(* IEC 61131-3 sources: moqui-plc/iec61131/moqui/runtime/component/mantle-hvac/src/main/org/moqui/device, 14 files *)

(* ---- AirDistributionControllerStatus.st ---- *)
TYPE AirDistributionControllerStatus : (
    Init := 0,
    HighPhase,
    TransitionToLow,
    LowPhase,
    TransitionToHigh
); END_TYPE

(* ---- DeviceFacade.dut ---- *)
(*#-#-#-#-#-#-#-#-#-#---Declaration---#-#-#-#-#-#-#-#-#-#-#-#-#*)

(*
 * DeviceFacade implementation for managing devices and logical parameters.
 *
 * Naming rules:
 *   deviceName + parameterName or parameterName → logical signal
 *   deviceName + parameterName or parameterName + Min/Max → limits
 *
 * All digital signals (boolean) are active-high (positive logic).
 * All durations are expressed in seconds TUnit.
 *)
TYPE DeviceFacade : STRUCT
	(* HVAC process control parameters (setpoints, limits, etc.) and process sensor signals *)
    (* Cell T+RH sensor  *)
    (* Setpoints and limits - mapped from recipe *)
    tempSetpoint : REAL; (* °C target process temperature *)
    tempHysteresis : REAL; (* °C symmetric hysteresis band *)
    tempMin : REAL;   (* °C absolute lower limit (alarm) *)
    tempMax : REAL; (* °C absolute upper limit (alarm) *)
    rhSetpoint : REAL; (* %  target relative humidity *)
    rhHysteresis : REAL; (* %  symmetric hysteresis band *)
    rhMin : REAL; (* % lower limit *)
    rhMax : REAL; (* % upper limit *)
    (* Core / surface probes - optional, used for thawing phases *)
    tempCoreSetpoint : REAL;
    tempCoreHysteresis : REAL;
    tempSurfaceSetpoint : REAL;
    tempSurfaceHysteresis : REAL;
    tempSurfaceMax : REAL;

    (* Feedback - wired from InputSignalUpdate each scan *)
    tempFeedback : REAL; (* °C cell air temperature *)
    rhFeedback : REAL; (* % cell relative humidity *)
    tempCoreFeedback : REAL; (* °C product core temperature *)
    tempSurfaceFeedback : REAL; (* °C product surface temperature *)

    (* Duct T+RH sensor (probe in the pipes) *)
    (* Limits - mapped from recipe or fixed commissioning values *)
    ductTempMin : REAL; (* °C minimum safe supply-air temperature *)
    ductTempMax : REAL; (* °C maximum safe supply-air temperature *)
    ductRhMax : REAL; (* % maximum allowed supply-air humidity *)
    (* Feedback - wired from InputSignalUpdate each scan *)
    ductTempFeedback : REAL; (* °C supply-air temperature in duct *)
    ductRhFeedback : REAL; (* % supply-air relative humidity in duct *)

    (* Boolean predicates - computed each scan by MainRuleEngine *)
    (* Cell sensor *)
    tempInRange : BOOL; (* tempMin+hys ≤ T ≤ tempMax-hys *)
    tempAtSetpoint : BOOL; (* |T - Tsp| ≤ hys *)
    tempOverMax : BOOL; (* T > tempMax *)
    tempOverMin : BOOL; (* T > tempMin *)
    tempUnderMin : BOOL; (* T < tempMin *)
    tempUnderMax : BOOL; (* T < tempMax *)
    tempCoreAtSetpoint : BOOL;
    tempSurfaceAtSetpoint : BOOL;
    tempSurfaceOverMax : BOOL;
    tempSurfaceUnderMax : BOOL;
    rhAtSetpoint : BOOL;
    rhOverMax  : BOOL; (* RH > rhMax - hys *)
    rhUnderMin : BOOL; (* RH < rhMin + hys *)
    rhOverMin : BOOL;
    rhUnderMax : BOOL;
    (* Duct sensor - safety predicates *)
    ductTempOverMax : BOOL; (* Supply air too hot → product at risk  *)
    ductTempUnderMin : BOOL; (* Supply air too cold → product at risk  *)
    ductRhOverMax : BOOL; (* Supply air saturated → condensation risk *)

    (* Operating-mode flags and process timing (mapped from recipe). *)
    rhControlEnabled : BOOL; (* Cooling+Heating both active for RH ctrl *)
    rhControlOnly : BOOL; (* Stop when RH ≤ rhMin regardless of time *)
    tempCoreControlEnabled : BOOL; (* Use core probe for thawing end-of-phase *)
    airMixingEnabled : BOOL;
    (* Process cycle durations (seconds) *)
    processEstimatedDuration : UDINT;
    processMinDuration : UDINT;
    processActualDuration : UDINT;
    processRemainingDuration : UDINT;
    (* Process time tracking *)
    (* Run / break cycle - phase 4 *)
    estimatedRuntime : UDINT;
    minRuntime : UDINT;
    actualRuntime : UDINT;
    estimatedBreakDuration : UDINT;
    minBreakDuration : UDINT;
    actualBreakDuration : UDINT;
    (* Air mixing sub-cycle *)
    airMixingEstimatedDuration : UDINT;
    airMixingMinDuration : UDINT;
    airMixingActualDuration : UDINT;
    airMixingEstimatedBreakDuration : UDINT;
    airMixingMinBreakDuration : UDINT;
    airMixingActualBreakDuration : UDINT;
    (* Flags *)
    (*
     * For operations based on equalization phases, rest/recovery periods are used,
     * during which moisture is evenly redistributed between the core
     * and the surface of the product after an intense drying phase (pulling).
     *)
    timeBreakEnabled : BOOL; (* TRUE while in break period *)
    isCompleted : BOOL; (* TRUE when the work effort is finished *)

    (* Main FSM state and transition request/acknowledge commands *)
    status : MainStatus := MainStatus.Standby;
    lastStatus : MainStatus := MainStatus.Standby;
    (*
     * Internally generated transition requests (set by MainRuleEngine,
     * consumed and cleared by Main.pou each scan)
     *)
    standbyRequest : BOOL;
    ventilationRequest : BOOL;
    coolingRequest : BOOL;
    heatingRequest : BOOL;
    dryingRequest : BOOL;
    surfaceThawingRequest : BOOL;
    coreThawingRequest : BOOL;
    faultRequest : BOOL;
    resetRequest : BOOL;

    (* HVAC devices *)

    (* Cold glycol group *)
    (* Enable/disable requests: written by Main component, read by DeviceManager *)
    coldGroupEnableRequest : BOOL;
    coldGroupDisableRequest : BOOL;
    (* Glycol circulating pump - on/off Actuator *)
    coldGlycolPump : Actuator;
    (* Modulating glycol valve - continuous PID control *)
    coldGlycolValve : ProcessPid;

    (* Hot glycol group *)
    hotGroupEnableRequest : BOOL;
    hotGroupDisableRequest : BOOL;
    hotGlycolPump : Actuator;
    hotGlycolValve : ProcessPid;

    (* AHU fan *)
    ahuFanEnableRequest : BOOL;
    (* Speed setpoint (0.0 … 100.0 %) - from recipe *)
    ahuFanSpeedSetpoint : REAL;
    (* Speed feedback (0.0 … 100.0 %) - from InputSignalUpdate *)
    ahuFanSpeedFeedback : REAL;
    ahuFan : ProcessPid;

    (* Air-flow distributor *)
    (* Treated as Actuator with additional ref/feedback.
     * The drive alternates air distribution between left and right ducts.
     * ref = time-split setpoint (0-100 %, 0 = full left, 100 = full right).
     * feedback = actual drive speed feedback.
	 *)
    airFlowEnableRequest : BOOL;
    airFlowDisableRequest : BOOL;
    airFlowRef : REAL; (* duty-cycle / distribution setpoint *)
    airFlowSpeedFeedback : REAL; (* drive speed feedback *)
    airFlow : Actuator;

    (* Signal management - centralised fault / alarm / warning engine *)
    signalMgmt : SignalMgmt;
END_STRUCT END_TYPE

(* ---- DeviceFacade.st ---- *)
(*
 * DeviceFacade implementation for managing devices and logical parameters.
 *
 * Naming rules:
 *   deviceName + parameterName or parameterName -> logical signal
 *   deviceName + parameterName or parameterName + Min/Max -> limits
 *
 * All digital signals (boolean) are active-high (positive logic).
 * All durations are expressed in seconds TUnit.
 *)
TYPE DeviceFacade : STRUCT
	(* HVAC process control parameters (setpoints, limits, etc.) and process sensor signals *)
    (* Cell T+RH sensor  *)
    (* Setpoints and limits - mapped from recipe *)
    tempSetpoint : REAL; (* °C target process temperature *)
    tempHysteresis : REAL; (* °C symmetric hysteresis band *)
    tempMin : REAL;   (* °C absolute lower limit (alarm) *)
    tempMax : REAL; (* °C absolute upper limit (alarm) *)
    rhSetpoint : REAL; (* %  target relative humidity *)
    rhHysteresis : REAL; (* %  symmetric hysteresis band *)
    rhMin : REAL; (* % lower limit *)
    rhMax : REAL; (* % upper limit *)
    (* Feedback - wired from InputSignalUpdate each scan *)
    tempFeedback : REAL; (* °C zone air temperature *)
    rhFeedback : REAL; (* % zone relative humidity *)

    (* Duct T+RH sensor (probe in the pipes) *)
    (* Limits - mapped from recipe or fixed commissioning values *)
    ductTempMin : REAL; (* °C minimum safe supply-air temperature *)
    ductTempMax : REAL; (* °C maximum safe supply-air temperature *)
    ductRhMax : REAL; (* % maximum allowed supply-air humidity *)
    (* Feedback - wired from InputSignalUpdate each scan *)
    ductTempFeedback : REAL; (* °C supply-air temperature in duct *)
    ductRhFeedback : REAL; (* % supply-air relative humidity in duct *)

    (* Boolean predicates - computed each scan by MainRuleEngine *)
    (* Cell sensor *)
    tempInRange : BOOL; (* tempMin+hys <= T <= tempMax-hys *)
    tempAtSetpoint : BOOL; (* |T - Tsp| <= hys *)
    tempAboveSetpointBand : BOOL; (* T >= tempSetpoint + tempHysteresis *)
    tempBelowSetpointBand : BOOL; (* T <= tempSetpoint - tempHysteresis *)
    tempOverMax : BOOL; (* T > tempMax *)
    tempOverMin : BOOL; (* T > tempMin *)
    tempUnderMin : BOOL; (* T < tempMin *)
    tempUnderMax : BOOL; (* T < tempMax *)
    rhAtSetpoint : BOOL;
    rhOverMax  : BOOL; (* RH > rhMax - hys *)
    rhUnderMin : BOOL; (* RH < rhMin + hys *)
    rhOverMin : BOOL;
    rhUnderMax : BOOL;
    (* Duct sensor - safety predicates *)
    ductTempOverMax : BOOL; (* Supply air too hot -> temperature limit violation *)
    ductTempUnderMin : BOOL; (* Supply air too cold -> temperature limit violation *)
    ductRhOverMax : BOOL; (* Supply air saturated -> condensation risk *)

    (* Operating-mode flags and process timing (mapped from recipe). *)
    rhControlEnabled : BOOL; (* Cooling+Heating both active for RH ctrl *)
    rhControlOnly : BOOL; (* Stop when RH <= rhMin regardless of time *)
    (* Air mixing *)
    airMixingEnabled : BOOL;
    airMixingFanEnableRequest : BOOL;
    airMixingFanDisableRequest : BOOL;
    airMixingFan : Actuator;
	(* Air distribution setpoints *)
	airDistributionEnabled : BOOL;
    setPointTimeHigh : UINT; (* Required cumulative time for high throw [s] *)
    setPointTimeLow : UINT; (* Required cumulative time for low throw [s] *)
    (* Process cycle durations (seconds) *)
    processEstimatedDuration : UDINT;
    processMinDuration : UDINT;
    processActualDuration : UDINT;
    processRemainingDuration : UDINT;
    (* Process time tracking *)
    (* Run / break cycle - Mode E *)
    estimatedRuntime : UDINT;
    minRuntime : UDINT;
    actualRuntime : UDINT;
    estimatedBreakDuration : UDINT;
    minBreakDuration : UDINT;
    actualBreakDuration : UDINT;
    (* Flags *)
    timeBreakEnabled : BOOL; (* TRUE while in break period *)
    isCompleted : BOOL; (* TRUE when the work effort is finished *)

    (* Main FSM state and transition request/acknowledge commands *)
    status : MainStatus := MainStatus.Standby;
    lastStatus : MainStatus := MainStatus.Standby;
    (*
     * Internally generated transition requests (set by MainRuleEngine,
     * consumed and cleared by Main.pou each scan)
     *)
    standbyRequest : BOOL;
    ventilationRequest : BOOL;
    coolingRequest : BOOL;
    heatingRequest : BOOL;
    dryingRequest : BOOL;
    faultRequest : BOOL;
    resetRequest : BOOL;

    (* HVAC devices *)

    (* Cold glycol group *)
    (* Enable/disable requests: written by Main component, read by DeviceManager *)
    coldGroupEnableRequest : BOOL;
    coldGroupDisableRequest : BOOL;
    (* Glycol circulating pump - on/off Actuator *)
    coldGlycolPump : Actuator;
    (* Modulating glycol valve - continuous PID control *)
    coldGlycolValve : ProcessPid;

    (* Hot glycol group *)
    hotGroupEnableRequest : BOOL;
    hotGroupDisableRequest : BOOL;
    hotGlycolPump : Actuator;
    hotGlycolValve : ProcessPid;

    (* AHU fan *)
    ahuFanEnableRequest : BOOL;
    (* Speed setpoint (0.0 … 100.0 %) - from recipe *)
    ahuFanSpeedSetpoint : REAL;
    (* Speed feedback (0.0 … 100.0 %) - from InputSignalUpdate *)
    ahuFanSpeedFeedback : REAL;
    ahuFan : ProcessPid;

    (* Air-flow distributor *)
    (* Treated as Actuator with additional ref/feedback.
     * The drive alternates air distribution between left and right ducts.
     * ref = time-split setpoint (0-100 %, 0 = full left, 100 = full right).
     * feedback = actual drive speed feedback.
	 *)
    airFlowEnableRequest : BOOL;
    airFlowDisableRequest : BOOL;
    airFlowRef : REAL; (* duty-cycle / distribution setpoint *)
    airFlowSpeedFeedback : REAL; (* drive speed feedback *)
    airFlow : Actuator;

    (* High flow damper *)
    highFlowDamperEnableRequest : BOOL;
    highFlowDamperDisableRequest : BOOL;
    highFlowDamper : Actuator;

    (* Low flow damper *)
    lowFlowDamperEnableRequest : BOOL;
    lowFlowDamperDisableRequest : BOOL;
    lowFlowDamper : Actuator;

    (* Signal management - centralised fault / alarm / warning engine *)
    signalMgmt : SignalMgmt;
END_STRUCT END_TYPE

(* ---- IOFacade.dut ---- *)
(*#-#-#-#-#-#-#-#-#-#---Declaration---#-#-#-#-#-#-#-#-#-#-#-#-#*)

(*
 * IOFacade implementation for managing physical devices and input/output signals/terminals.
 * Input/Output physical terminals naming rules.
 * From each value of the Parameter entity 3 signals will be generated, according to the following naming convention:
 *     deviceName + parameterName or parameterName + physicalAddress (e.g.: Channel + PhysicalAddress for Modbus)
 * 	   deviceName + parameterName or parameterName + Min/Max + physicalAddress (e.g.: Channel + PhysicalAddress for Modbus)
 *
 * The physicalAdddress suffix will have the following syntax:
	   %<memory area prefix> ( <size prefix> )? <memory position>
 * where
 * 	   <memory area prefix> : I | Q | M
 *     <size prefix> : X | B | W | D
 *     <memory position> : <number> ( .<number> )* (* Depends on the target system *)
 *
 * An alternative is to use the following semantic signal naming rules:
 *
 *     (* AHU fan physical input signals *)
 *     ahuFanDriveControlWord : WORD;
 *     ahuFanDriveStatusWord : WORD;
 *     ahuFanDriveRO1 : BOOL; (* Relay output 1 *)
 *
 *     (* Air renewal fan physical input signals *)
 *     airRenewalFanDriveControlWord : WORD;
 *     airRenewalFanDriveStatusWord : WORD;
 *     airRenewalFanDriveRO1 : BOOL; (* Relay output 1 *)
 *
 *     (* Cold glycol circulating pump physical input signals *)
 *     coldGlycolPumpMotorStarterSignalingContact : BOOL;
 *     coldGlycolPumpMotorStarterShuntTrip : BOOL;
 *     coldGlycolPumpContactorSignalingContact : BOOL;
 *
 *     ...
 *
 *)
TYPE IOFacade : STRUCT
	(* ========== Phyisical Input Terminals/Signals ========== *)

	(* Motion example: *)
	speedFeedbackSignal : ARRAY[0..1] OF WORD;
	accelerationFeedbackSignal : ARRAY[0..3] OF WORD;

	(* ========== Phyisical Output Terminals/Signals ========== *)

	(*
	(* Motion example: *)
	(* Example mapping for a word analog signal *)
    speedRefSignal : WORD;
	(* Example mapping for a 32-bit analog signal *)
    speedRefSignal : ARRAY[0..1] OF WORD;
	(* Example of an alternative mapping for a 64-bit analog signal *)
	speedRefSignal : ARRAY[0..3] OF WORD;
	(* Example of an alternative mapping for a 32-bit physical value to a REAL variable *)
	speedRefSignal : REAL;
	(* Example of an alternative mapping for a 64-bit physical value to an LREAL variable *)
	speedRefSignal : REAL;
	(* It is possible to apply the same logic to other variables such as: acceleration/deceleration, torque, etc. *)
	*)

	(* ABB IO remote device information *)
	io1DeviceInformationBlock : WORD;
END_STRUCT END_TYPE

(* ---- IOFacade.st ---- *)
(*
 * IOFacade implementation for managing physical devices and input/output signals/terminals.
 * Input/Output physical terminals naming rules.
 * From each value of the Parameter entity 3 signals will be generated, according to the following naming convention:
 *     deviceName + parameterName or parameterName + physicalAddress (e.g.: Channel + PhysicalAddress for Modbus)
 * 	   deviceName + parameterName or parameterName + Min/Max + physicalAddress (e.g.: Channel + PhysicalAddress for Modbus)
 *
 * The physicalAdddress suffix will have the following syntax:
	   %<memory area prefix> ( <size prefix> )? <memory position>
 * where
 * 	   <memory area prefix> : I | Q | M
 *     <size prefix> : X | B | W | D
 *     <memory position> : <number> ( .<number> )* (* Depends on the target system *)
 *
 * An alternative is to use the following semantic signal naming rules:
 *
 *     (* AHU fan physical input signals *)
 *     ahuFanDriveControlWord : WORD;
 *     ahuFanDriveStatusWord : WORD;
 *     ahuFanDriveRO1 : BOOL; (* Relay output 1 *)
 *
 *     (* Air renewal fan physical input signals *)
 *     airRenewalFanDriveControlWord : WORD;
 *     airRenewalFanDriveStatusWord : WORD;
 *     airRenewalFanDriveRO1 : BOOL; (* Relay output 1 *)
 *
 *     (* Cold glycol circulating pump physical input signals *)
 *     coldGlycolPumpMotorStarterSignalingContact : BOOL;
 *     coldGlycolPumpMotorStarterShuntTrip : BOOL;
 *     coldGlycolPumpContactorSignalingContact : BOOL;
 *
 *     ...
 *
 *)
TYPE IOFacade : STRUCT
	(* ========== Phyisical Input Terminals/Signals ========== *)

	(* Motion example: *)
	speedFeedbackSignal : ARRAY[0..1] OF WORD;
	accelerationFeedbackSignal : ARRAY[0..3] OF WORD;

	(* ========== Phyisical Output Terminals/Signals ========== *)

	(*
	(* Motion example: *)
	(* Example mapping for a word analog signal *)
    speedRefSignal : WORD;
	(* Example mapping for a 32-bit analog signal *)
    speedRefSignal : ARRAY[0..1] OF WORD;
	(* Example of an alternative mapping for a 64-bit analog signal *)
	speedRefSignal : ARRAY[0..3] OF WORD;
	(* Example of an alternative mapping for a 32-bit physical value to a REAL variable *)
	speedRefSignal : REAL;
	(* Example of an alternative mapping for a 64-bit physical value to an LREAL variable *)
	speedRefSignal : REAL;
	(* It is possible to apply the same logic to other variables such as: acceleration/deceleration, torque, etc. *)
	*)

	(* ABB IO remote device information *)
	io1DeviceInformationBlock : WORD;
END_STRUCT END_TYPE

(* ---- AirDistributionController.st ---- *)
(*
 * AirDistributionController: Logical sequencer for alternating high/low air throw.
 *
 * Implements cumulative timing logic for throw phases:
 * - Time advances only during active operation (operationType = Run AND enable = TRUE).
 * - Counters are frozen (retained) during standby/pause phases.
 * - Implements a Make-Before-Break transition between ducts to prevent overpressure peaks,
 * leveraging the asynchronous handshake mechanism (VAR_IN_OUT) of the underlying Actuator instances.
 *)
FUNCTION_BLOCK AirDistributionController
	VAR_EXTERNAL
	    dev : DeviceFacade;
	END_VAR
	VAR_INPUT
	    operationType : OperatingMode := OperatingMode.Init;
	    enable : BOOL; (* Local run permission (e.g., air flow running + air mixing enabled) *)
	    clock1s : BOOL; (* 1-second base clock pulse *)
	END_VAR
	VAR CONSTANT
	    componentName : STRING := 'HVAC_AIR_GROUP';
	END_VAR
	VAR
		(* Logger facade *)
	    logger : LoggerFacade;
	    status : AirDistributionControllerStatus := AirDistributionControllerStatus.Init;
	    cumulatedTimeHigh : UINT := 0;
	    cumulatedTimeLow : UINT := 0;
	END_VAR

	(* Logger facade init *)
	logger.enable := TRUE; logger.loggerName := componentName;

	(* Initialization or reset upon critical Stop *)
	IF operationType = OperatingMode.Init THEN
	    logger(message := 'Init air distribution controller.', level := LogLevel.DEBUG);
	    status := AirDistributionControllerStatus.Init;
	    cumulatedTimeHigh := 0;
	    cumulatedTimeLow := 0;
		dev.highFlowDamperEnableRequest := TRUE;
		dev.highFlowDamperDisableRequest := FALSE;
		dev.lowFlowDamperEnableRequest := FALSE;
		dev.lowFlowDamperDisableRequest := TRUE;
	    RETURN;
	END_IF;

	(* Logic advances ONLY if the system is in Run mode and local enable is active *)
	IF (operationType = OperatingMode.Run) AND enable THEN

	    CASE status OF

	        AirDistributionControllerStatus.Init:
	            (* Startup sequence: defaults to the high throw phase *)
	            dev.highFlowDamperEnableRequest := TRUE;
	 		   	dev.highFlowDamperDisableRequest := FALSE;
	            dev.lowFlowDamperEnableRequest := FALSE;
	 		   	dev.lowFlowDamperDisableRequest := TRUE;
	            logger(message := 'Enter high throw phase.', level := LogLevel.DEBUG);
	            status := AirDistributionControllerStatus.HighPhase;

	        AirDistributionControllerStatus.HighPhase:
	            (* Advance cumulative timer *)
	            IF clock1s THEN
	                cumulatedTimeHigh := cumulatedTimeHigh + 1;
	            END_IF;

	            (* Evaluate switching threshold *)
	            IF dev.setPointTimeHigh > 0 AND cumulatedTimeHigh >= dev.setPointTimeHigh THEN
	                cumulatedTimeHigh := 0;
	                (* Make-Before-Break Interlock / Asynchronous Handshake *)
					dev.highFlowDamperEnableRequest := FALSE;
					dev.highFlowDamperDisableRequest := TRUE;
					dev.lowFlowDamperEnableRequest := TRUE;
					dev.lowFlowDamperDisableRequest := FALSE;
	                logger(message := 'Transition to low throw.', level := LogLevel.DEBUG);
	                status := AirDistributionControllerStatus.TransitionToLow;
	            END_IF;

	        AirDistributionControllerStatus.TransitionToLow:
	            (* * Monitor the falling edge of the request signals.
	             * The Actuator block internally clears the VAR_IN_OUT variable once
	             * the physical maneuver is completed. This ensures the sequencer
	             * advances only after the hardware has reached its target position.
	             *)
	            IF NOT dev.highFlowDamperDisableRequest AND NOT dev.lowFlowDamperEnableRequest THEN
	                logger(message := 'Enter low throw phase.', level := LogLevel.DEBUG);
	                status := AirDistributionControllerStatus.LowPhase;
	            END_IF;

	        AirDistributionControllerStatus.LowPhase:
	            (* Advance cumulative timer *)
	            IF clock1s THEN
	                cumulatedTimeLow := cumulatedTimeLow + 1;
	            END_IF;

	            (* Evaluate switching threshold *)
	            IF dev.setPointTimeLow > 0 AND cumulatedTimeLow >= dev.setPointTimeLow THEN
	                cumulatedTimeLow := 0;
	                (* Make-Before-Break Interlock / Asynchronous Handshake *)
					dev.highFlowDamperEnableRequest := TRUE;
					dev.highFlowDamperDisableRequest := FALSE;
					dev.lowFlowDamperEnableRequest := FALSE;
					dev.lowFlowDamperDisableRequest := TRUE;
	                logger(message := 'Transition to high throw.', level := LogLevel.DEBUG);
	                status := AirDistributionControllerStatus.TransitionToHigh;
	            END_IF;

	        AirDistributionControllerStatus.TransitionToHigh:
	            (* Wait for hardware positioning confirmation *)
	            IF NOT dev.lowFlowDamperDisableRequest AND NOT dev.highFlowDamperEnableRequest THEN
	                logger(message := 'Enter high throw phase.', level := LogLevel.DEBUG);
	                status := AirDistributionControllerStatus.HighPhase;
	            END_IF;
	    END_CASE;
	ELSE
	    (* Standby / Pause Condition *)
	    (*
	     * During standby (OperatingMode.Standby OR enable = FALSE), the FB does
	     * not increment any timers. The current status and Request variables are
	     * frozen, maintaining the hardware in its last consolidated stable state.
	     *)
	    ;
	END_IF;
	END_FUNCTION_BLOCK

(* ---- DeviceDiagnostics.pou ---- *)
(*#-#-#-#-#-#-#-#-#-#---Declaration---#-#-#-#-#-#-#-#-#-#-#-#-#*)

{attribute 'no_assign'}
(* Device diagnostics *)
FUNCTION_BLOCK DeviceDiagnostics
VAR_EXTERNAL
	dev : DeviceFacade;
END_VAR
VAR_INPUT
	operationType : OperatingMode := OperatingMode.Run;
END_VAR
VAR_OUTPUT
	error : BOOL;
END_VAR

(*#-#-#-#-#-#-#-#-#-#---Implementation---#-#-#-#-#-#-#-#-#-#-#-#-#*)

error := TRUE;

(* Signal management engine *)
(*
 * Prepare a fresh scan (clears the accumulated output action).
 * Then process each device signal in priority order.
 * ImmediateStop → faultRequest := TRUE → Main enters Fault state.
 *)
dev.signalMgmt(operationType := SignalMgmtOperatingMode.Prepare);
dev.signalMgmt.operationType := SignalMgmtOperatingMode.Process;

(* Device faults *)
dev.signalMgmt(
	loggerName := dev.ahuFan.loggerName,
	code := 16#0001,
	category := SignalCategory.Alarm,
	resetPol := ResetPolicy.UnconditionedReset,
	activationCondition := dev.ahuFan.invalidConfig,
	outputAction := SignalOutputAction.ImmediateStop);
dev.signalMgmt(
	loggerName := dev.airFlow.loggerName,
	code := 16#0002,
	category := SignalCategory.Alarm,
	resetPol := ResetPolicy.UnconditionedReset,
	activationCondition := dev.airFlow.fault,
	outputAction := SignalOutputAction.ImmediateStop);
dev.signalMgmt(
	loggerName := dev.coldGlycolPump.loggerName,
	code := 16#0003,
	category := SignalCategory.Alarm,
	resetPol := ResetPolicy.UnconditionedReset,
	activationCondition := dev.coldGlycolPump.fault,
	outputAction := SignalOutputAction.ImmediateStop);
dev.signalMgmt(
	loggerName := dev.coldGlycolValve.loggerName,
	code := 16#0004,
	category := SignalCategory.Alarm,
	resetPol := ResetPolicy.UnconditionedReset,
	activationCondition := dev.coldGlycolValve.invalidConfig,
	outputAction := SignalOutputAction.ImmediateStop);
dev.signalMgmt(
	loggerName := dev.hotGlycolPump.loggerName,
	code := 16#0005,
	category := SignalCategory.Alarm,
	resetPol := ResetPolicy.UnconditionedReset,
	activationCondition := dev.hotGlycolPump.fault,
	outputAction := SignalOutputAction.ImmediateStop);
dev.signalMgmt(
	loggerName := dev.hotGlycolValve.loggerName,
	code := 16#0006,
	category := SignalCategory.Alarm,
	resetPol := ResetPolicy.UnconditionedReset,
	activationCondition := dev.hotGlycolValve.invalidConfig,
	outputAction := SignalOutputAction.ImmediateStop);

(*
 * Duct safety alarms - supply-air temperature limits (ImmediateStop).
 * Air that is too hot or too cold entering the curing room can damage
 * or contaminate the product. These alarms are always evaluated
 * regardless of the current FSM state.
 *)
dev.signalMgmt(
	loggerName := 'ductSensor',
	code := 16#0010,
	category := SignalCategory.Alarm,
	resetPol := ResetPolicy.UnconditionedReset,
	activationCondition := dev.ductTempOverMax,
	outputAction := SignalOutputAction.ImmediateStop);
dev.signalMgmt(
	loggerName := 'ductSensor',
	code := 16#0011,
	category := SignalCategory.Alarm,
	resetPol := ResetPolicy.UnconditionedReset,
	activationCondition := dev.ductTempUnderMin,
	outputAction := SignalOutputAction.ImmediateStop);

(* Duct RH - Warning only (condensation risk, does not stop the machine) *)
dev.signalMgmt(
	loggerName := 'ductSensor',
	code := 16#0012,
	category := SignalCategory.Warning,
	resetPol := ResetPolicy.UnconditionedReset,
	activationCondition := dev.ductRhOverMax,
	outputAction := SignalOutputAction.None);

error := FALSE;

(* ---- DeviceDiagnostics.st ---- *)
(* Device diagnostics *)
FUNCTION_BLOCK DeviceDiagnostics
	VAR_EXTERNAL
		dev : DeviceFacade;
	END_VAR
	VAR_INPUT
		operationType : OperatingMode := OperatingMode.Run;
	END_VAR
	VAR_OUTPUT
		error : BOOL;
	END_VAR

	error := TRUE;

	(* Signal management engine *)
	(*
	 * Prepare a fresh scan (clears the accumulated output action).
	 * Then process each device signal in priority order.
	 * ImmediateStop -> faultRequest := TRUE -> Main enters Fault state.
	 *)
	dev.signalMgmt(operationType := SignalMgmtOperatingMode.Prepare);
	dev.signalMgmt.operationType := SignalMgmtOperatingMode.Process;

	(* Device faults *)
	dev.signalMgmt(
		loggerName := dev.ahuFan.loggerName,
		code := 16#0001,
		category := SignalCategory.Alarm,
		resetPol := ResetPolicy.UnconditionedReset,
		activationCondition := dev.ahuFan.invalidConfig,
		outputAction := SignalOutputAction.ImmediateStop);
	dev.signalMgmt(
		loggerName := dev.airFlow.loggerName,
		code := 16#0002,
		category := SignalCategory.Alarm,
		resetPol := ResetPolicy.UnconditionedReset,
		activationCondition := dev.airFlow.fault,
		outputAction := SignalOutputAction.ImmediateStop);
	dev.signalMgmt(
		loggerName := dev.coldGlycolPump.loggerName,
		code := 16#0003,
		category := SignalCategory.Alarm,
		resetPol := ResetPolicy.UnconditionedReset,
		activationCondition := dev.coldGlycolPump.fault,
		outputAction := SignalOutputAction.ImmediateStop);
	dev.signalMgmt(
		loggerName := dev.coldGlycolValve.loggerName,
		code := 16#0004,
		category := SignalCategory.Alarm,
		resetPol := ResetPolicy.UnconditionedReset,
		activationCondition := dev.coldGlycolValve.invalidConfig,
		outputAction := SignalOutputAction.ImmediateStop);
	dev.signalMgmt(
		loggerName := dev.hotGlycolPump.loggerName,
		code := 16#0005,
		category := SignalCategory.Alarm,
		resetPol := ResetPolicy.UnconditionedReset,
		activationCondition := dev.hotGlycolPump.fault,
		outputAction := SignalOutputAction.ImmediateStop);
	dev.signalMgmt(
		loggerName := dev.hotGlycolValve.loggerName,
		code := 16#0006,
		category := SignalCategory.Alarm,
		resetPol := ResetPolicy.UnconditionedReset,
		activationCondition := dev.hotGlycolValve.invalidConfig,
		outputAction := SignalOutputAction.ImmediateStop);
	dev.signalMgmt(
		loggerName := dev.highFlowDamper.loggerName,
		code := 16#0007,
		category := SignalCategory.Alarm,
		resetPol := ResetPolicy.UnconditionedReset,
		activationCondition := dev.highFlowDamper.fault,
		outputAction := SignalOutputAction.ImmediateStop);
	dev.signalMgmt(
		loggerName := dev.lowFlowDamper.loggerName,
		code := 16#0008,
		category := SignalCategory.Alarm,
		resetPol := ResetPolicy.UnconditionedReset,
		activationCondition := dev.lowFlowDamper.fault,
		outputAction := SignalOutputAction.ImmediateStop);

	(*
	 * Duct safety alarms - supply-air temperature limits (ImmediateStop).
	 * Air that is too hot or too cold entering the curing room can damage
	 * or contaminate the product. These alarms are always evaluated
	 * regardless of the current FSM state.
	 *)
	dev.signalMgmt(
		loggerName := 'HVAC_DEMO_PLC',
		code := 16#0010,
		category := SignalCategory.Alarm,
		resetPol := ResetPolicy.UnconditionedReset,
		activationCondition := dev.ductTempOverMax,
		outputAction := SignalOutputAction.ImmediateStop);
	dev.signalMgmt(
		loggerName := 'HVAC_DEMO_PLC',
		code := 16#0011,
		category := SignalCategory.Alarm,
		resetPol := ResetPolicy.UnconditionedReset,
		activationCondition := dev.ductTempUnderMin,
		outputAction := SignalOutputAction.ImmediateStop);

	(* Duct RH - Warning only (condensation risk, does not stop the machine) *)
	dev.signalMgmt(
		loggerName := 'HVAC_DEMO_PLC',
		code := 16#0012,
		category := SignalCategory.Warning,
		resetPol := ResetPolicy.UnconditionedReset,
		activationCondition := dev.ductRhOverMax,
		outputAction := SignalOutputAction.None);

	error := FALSE;
	END_FUNCTION_BLOCK

(* ---- DeviceManager.pou ---- *)
(*#-#-#-#-#-#-#-#-#-#---Declaration---#-#-#-#-#-#-#-#-#-#-#-#-#*)

{attribute 'no_assign'}
(* Hardware Abstraction Layer (HAL) orchestrator.
 *
 * Drives all physical device FBs once per scan.
 * Main component sets the enable/disable request flags; DeviceManager wires them
 * to the individual Actuator / ActuatorGroup / ProcessPid / Axis / AxisGroup FBs.
 *
 * Call order within the PLC task:
 *   InputSignalUpdate (updates feedback signals from field)
 *   Main (FSM + MainRuleEngine → sets request flags)
 *   DeviceManager (this block - drives device FBs)
 *   OutputSignalUpdate (maps device outputs to physical terminals)
 *
 * Handshake note (Actuator FBs):
 *   enableRequest / disableRequest are VAR_IN_OUT.  The Actuator FB clears
 *   the flag as its acknowledgment.  Main.pou re-asserts the flag each scan
 *   from dev.xxxEnableRequest, so the handshake is level-triggered.
 *
 * ProcessPid note (ahuFan):
 *   ProcessPid uses a plain BOOL 'enable' input - no VAR_IN_OUT handshake.
 *   Setting enable := FALSE ramps the output to 0 and disables the controller.
 *)
FUNCTION_BLOCK DeviceManager
VAR_EXTERNAL
	clks : Clocks;
	dev : DeviceFacade;
END_VAR
VAR_INPUT
	operationType : OperatingMode := OperatingMode.Run;
END_VAR

(*#-#-#-#-#-#-#-#-#-#---Implementation---#-#-#-#-#-#-#-#-#-#-#-#-#*)

(* Cold glycol group *)
(*
 * Pump is started first via the request/ack handshake.
 * Valve enable follows the group request directly (no separate handshake
 * needed for ProcessPid - enable := FALSE freezes the output at 0).
 *)
dev.coldGlycolPump(
	operationType := operationType,
	clock := clks.clock100ms,
	enableRequest := dev.coldGroupEnableRequest,
	disableRequest := dev.coldGroupDisableRequest);

dev.coldGlycolValve(
	enable := dev.coldGroupEnableRequest,
	feedback := dev.tempFeedback,
	setpoint := dev.tempSetpoint,
	clock := clks.clock100ms);

(* Hot glycol group *)
dev.hotGlycolPump(
	operationType := operationType,
	clock := clks.clock100ms,
	enableRequest := dev.hotGroupEnableRequest,
	disableRequest := dev.hotGroupDisableRequest);

dev.hotGlycolValve(
	enable := dev.hotGroupEnableRequest,
	feedback := dev.tempFeedback,
	setpoint := dev.tempSetpoint,
	clock := clks.clock100ms);

(* AHU fan *)
(*
 * enable := FALSE ramps down the drive and disables the PID output.
 * Speed setpoint (ahuFanSpeedSetpoint) and the PID tuning parameters
 * (gain, integrationTime, etc.) are mapped from the device config (recipe).
 * ahuFanSpeedFeedback is wired from InputSignalUpdate (drive feedback word).
 *)
dev.ahuFan(
	enable := dev.ahuFanEnableRequest,
	setpoint := dev.ahuFanSpeedSetpoint,
	feedback := dev.ahuFanSpeedFeedback,
	clock := clks.clock100ms);

(* Air flow distributor (drive) *)
(*
 * Treated as Actuator with an additional speed reference.
 * ref = distribution setpoint (0-100 %) from device config (recipe)/RuleEngine.
 * feedback = drive speed feedback from InputSignalUpdate.
 * The drive alternates supply air between left and right ducts
 * according to the ref timing programmed on the drive itself;
 * the PLC only starts / stops it and adjusts the reference level.
 *)
dev.airFlow(
	operationType := operationType,
	clock := clks.clock100ms,
	enableRequest := dev.airFlowEnableRequest,
	disableRequest := dev.airFlowDisableRequest,
	ref := dev.airFlowRef,
	feedback := dev.airFlowSpeedFeedback);

(* ---- DeviceManager.st ---- *)
(* Hardware Abstraction Layer (HAL) orchestrator.
 *
 * Drives all physical device FBs once per scan.
 * Main component sets the enable/disable request flags; DeviceManager wires them
 * to the individual Actuator / ProcessPid FBs.
 *
 * Call order within the PLC task:
 *   InputSignalUpdate (updates feedback signals from field)
 *   Main (FSM + MainRuleEngine -> sets request flags)
 *   DeviceManager (this block - drives device FBs)
 *   OutputSignalUpdate (maps device outputs to physical terminals)
 *
 * Handshake note (Actuator FBs):
 *   enableRequest / disableRequest are VAR_IN_OUT.  The Actuator FB clears
 *   the flag as its acknowledgment.  Main.pou re-asserts the flag each scan
 *   from dev.xxxEnableRequest, so the handshake is level-triggered.
 *
 * ProcessPid note (ahuFan):
 *   ProcessPid uses a plain BOOL 'enable' input - no VAR_IN_OUT handshake.
 *   Setting enable := FALSE ramps the output to 0 and disables the controller.
 *)
FUNCTION_BLOCK DeviceManager
	VAR_EXTERNAL
		clks : Clocks;
		dev : DeviceFacade;
	END_VAR
	VAR_INPUT
		operationType : OperatingMode := OperatingMode.Run;
	END_VAR

	(* Cold glycol group *)
	(*
	 * Pump is started first via the request/ack handshake.
	 * Valve enable follows the group request directly (no separate handshake
	 * needed for ProcessPid - enable := FALSE freezes the output at 0).
	 *)
	dev.coldGlycolPump(
		operationType := operationType,
		clock := clks.clock100ms,
		enableRequest := dev.coldGroupEnableRequest,
		disableRequest := dev.coldGroupDisableRequest);

	dev.coldGlycolValve(
		enable := dev.coldGroupEnableRequest,
		feedback := dev.tempFeedback,
		setpoint := dev.tempSetpoint,
		clock := clks.clock100ms);

	(* Hot glycol group *)
	dev.hotGlycolPump(
		operationType := operationType,
		clock := clks.clock100ms,
		enableRequest := dev.hotGroupEnableRequest,
		disableRequest := dev.hotGroupDisableRequest);

	dev.hotGlycolValve(
		enable := dev.hotGroupEnableRequest,
		feedback := dev.tempFeedback,
		setpoint := dev.tempSetpoint,
		clock := clks.clock100ms);

	(* AHU fan *)
	(*
	 * enable := FALSE ramps down the drive and disables the PID output.
	 * Speed setpoint (ahuFanSpeedSetpoint) and the PID tuning parameters
	 * (gain, integrationTime, etc.) are mapped from the device config (recipe).
	 * ahuFanSpeedFeedback is wired from InputSignalUpdate (drive feedback word).
	 *)
	dev.ahuFan(
		enable := dev.ahuFanEnableRequest,
		setpoint := dev.ahuFanSpeedSetpoint,
		feedback := dev.ahuFanSpeedFeedback,
		clock := clks.clock100ms);

	(* Air flow distributor (drive) *)
	(*
	 * Treated as Actuator with an additional speed reference.
	 * ref = distribution setpoint (0-100 %) from device config (recipe)/RuleEngine.
	 * feedback = drive speed feedback from InputSignalUpdate.
	 * The drive alternates supply air between left and right ducts
	 * according to the ref timing programmed on the drive itself;
	 * the PLC only starts / stops it and adjusts the reference level.
	 *)
	dev.airFlow(
		operationType := operationType,
		clock := clks.clock100ms,
		enableRequest := dev.airFlowEnableRequest,
		disableRequest := dev.airFlowDisableRequest,
		ref := dev.airFlowRef,
		feedback := dev.airFlowSpeedFeedback);

	(* High Flow Damper *)
	(* Requests are generated by AirDistributionController when air mixing is enabled. *)
	dev.highFlowDamper(
		operationType := operationType,
		clock := clks.clock100ms,
		enableRequest := dev.highFlowDamperEnableRequest,
		disableRequest := dev.highFlowDamperDisableRequest);

	(* Low Flow Damper *)
	(* Requests are generated by AirDistributionController when air mixing is enabled. *)
	dev.lowFlowDamper(
		operationType := operationType,
		clock := clks.clock100ms,
		enableRequest := dev.lowFlowDamperEnableRequest,
		disableRequest := dev.lowFlowDamperDisableRequest);
	END_FUNCTION_BLOCK

(* ---- InputSignalUpdate.pou ---- *)
(*#-#-#-#-#-#-#-#-#-#---Declaration---#-#-#-#-#-#-#-#-#-#-#-#-#*)

{attribute 'no_assign'}
(*
 * Input signal acquisition and pre-processing unit.
 * Map physical input terminals/signals to their logical parameters, performing pre-processing (e.g.: signal filtering) if necessary.
 *)
FUNCTION_BLOCK InputSignalUpdate
VAR_EXTERNAL
	dev : DeviceFacade;
	io : IOFacade;
END_VAR
VAR_INPUT
	operationType : OperatingMode;
END_VAR
VAR
	(* Logger facade *)
	logger : LoggerFacade;
END_VAR

(*#-#-#-#-#-#-#-#-#-#---Implementation---#-#-#-#-#-#-#-#-#-#-#-#-#*)

(* Logger facade init *)
logger.enable := TRUE; logger.loggerName := 'InputSignalUpdate';

logger(message := 'Input signals acquisition and pre-processing.', level := LogLevel.DEBUG);

(*
	Physical to logical terminals mapping example:

	IF operationType = OperatingMode.Init THEN
		(* Special processing for the init phase, if needed, such as the restart phase after a blackout. *)
		(* etc. *)
	ELSIF operationType = OperatingMode.Run THEN
		(* Example mapping of 32 bits and 64 bits analog signals *)
		dev.speedFeedback := doubleWordToReal(wordArray := io.speedFeedbackSignal);
		dev.speedFeedback := longWordToLongReal(wordArray := io.speedFeedbackSignal);
		(* Reverse logic *)
		dev.coldGlycolValve.disabledSensor := NOT io.coldGlycolValveSignalingContact;

		outletColdGlycolTemp := TO_REAL(outletColdGlycolTempSignal);
		(* Analog input processing (scaling, limiting, etc. *)
		dev.tempFeedback := processAnalogInput(io.tempFeedbackSignal, 0, 27000, dev.tempMin, dev.tempMax, -20, 70, 0);
		(* Analog input exponential (1-pole) filtering *)
		expFilter(input := io.coldGlycolTempSignal, t:= 3, start := TRUE, timeElapsed => timeElapsed);
		IF timeElapsed >= 3 THEN dev.outletColdGlycolTemp := expFilter.output; END_IF;
		(* Digital input processing (filtering, debouncing, reverse logic, etc. *)
		digitalFilter(signal := io.airFlowEnabledSensor, enableDelay := T#10MS, disableDelay := T#15MS);
		dev.airFlow.enabledSensor := digitalFilter.delayedSignal;
		(* Drive status word, feedbacks, etc. mapping *)
		processDriveCyclicInData(model := DriveModel.ABBACH580, statusWord := io.compressorStatusWord,
			enabledSensor => dev.compressor.enabledSensor, disabledSensor => dev.compressor.disabledSensor,
			externalFault => dev.compressorExternalFault);
		dev.speedFeedback := TO_REAL(speedFeedbackSignal);
		dev.coldGlycolPump.enabledSensor := io.coldGlycolPumpAuxContact;
		dev.coldGlycolPump.disabledSensor := NOT io.coldGlycolPumpAuxContact;
		dev.coldGlycolPumpThermistors := io.coldGlycolPumpThermistors;
		dev.coldGlycolFlowSwitch := io.coldGlycolFlowSwitch;
		dev.coldGlycolPumpPowerSupplyFault := NOT io.coldGlycolPumpShuntTrip;
		dev.coldGlycolCircPumpExternalFault := io.coldGlycolPumpShuntTrip OR io.coldGlycolPumpThermistors
			OR io.coldGlycolFlowSwitch;
		...

	END_IF;

	(*
	 * Configure and call the logger facade to log signals where needed.
	 *     logger(payloadType := LogPayloadType.Numeric, numericValue := dev.speedRef, level := LogLevel.DEBUG);
	 *     logger(payloadType := LogPayloadType.Numeric, numericValue := dev.outletColdGlycolTemp, level := LogLevel.DEBUG);
	 *     (* etc. *)
	 *)
*)

(* ---- InputSignalUpdate.st ---- *)
(*
 * Input signal acquisition and pre-processing unit.
 * Map physical input terminals/signals to their logical parameters, performing pre-processing (e.g.: signal filtering) if necessary.
 *)
FUNCTION_BLOCK InputSignalUpdate
	VAR_EXTERNAL CONSTANT
		applicationDeviceId : STRING;
	END_VAR
	VAR_EXTERNAL
		dev : DeviceFacade;
		io : IOFacade;
	END_VAR
	VAR_INPUT
		operationType : OperatingMode;
	END_VAR
	VAR
		(* Logger facade *)
		logger : LoggerFacade;
	END_VAR

	(* Logger facade init *)
	logger.enable := TRUE; logger.loggerName := applicationDeviceId;

	logger(message := 'Input signals acquisition and pre-processing.', level := LogLevel.DEBUG);

	(*
		Physical to logical terminals mapping example:

		IF operationType = OperatingMode.Init THEN
			(* Special processing for the init phase, if needed, such as the restart phase after a blackout. *)
			(* etc. *)
		ELSIF operationType = OperatingMode.Run THEN
			(* Example mapping of 32 bits and 64 bits analog signals *)
			dev.speedFeedback := doubleWordToReal(wordArray := io.speedFeedbackSignal);
			dev.speedFeedback := longWordToLongReal(wordArray := io.speedFeedbackSignal);
			(* Reverse logic *)
			dev.coldGlycolValve.disabledSensor := NOT io.coldGlycolValveSignalingContact;

			outletColdGlycolTemp := TO_REAL(outletColdGlycolTempSignal);
			(* Analog input processing (scaling, limiting, etc. *)
			dev.tempFeedback := processAnalogInput(io.tempFeedbackSignal, 0, 27000, dev.tempMin, dev.tempMax, -20, 70, 0);
			(* Analog input exponential (1-pole) filtering *)
			expFilter(input := io.coldGlycolTempSignal, t:= 3, start := TRUE, timeElapsed => timeElapsed);
			IF timeElapsed >= 3 THEN dev.outletColdGlycolTemp := expFilter.output; END_IF;
			(* Digital input processing (filtering, debouncing, reverse logic, etc. *)
			digitalFilter(signal := io.airFlowEnabledSensor, enableDelay := T#10MS, disableDelay := T#15MS);
			dev.airFlow.enabledSensor := digitalFilter.delayedSignal;
			(* Drive status word, feedbacks, etc. mapping *)
			processDriveCyclicInData(model := DriveModel.ABBACH580, statusWord := io.compressorStatusWord,
				enabledSensor => dev.compressor.enabledSensor, disabledSensor => dev.compressor.disabledSensor,
				externalFault => dev.compressorExternalFault);
			dev.speedFeedback := TO_REAL(speedFeedbackSignal);
			dev.coldGlycolPump.enabledSensor := io.coldGlycolPumpAuxContact;
			dev.coldGlycolPump.disabledSensor := NOT io.coldGlycolPumpAuxContact;
			dev.coldGlycolPumpThermistors := io.coldGlycolPumpThermistors;
			dev.coldGlycolFlowSwitch := io.coldGlycolFlowSwitch;
			dev.coldGlycolPumpPowerSupplyFault := NOT io.coldGlycolPumpShuntTrip;
			dev.coldGlycolCircPumpExternalFault := io.coldGlycolPumpShuntTrip OR io.coldGlycolPumpThermistors
				OR io.coldGlycolFlowSwitch;
			...

		END_IF;

		(*
		 * Configure and call the logger facade to log signals where needed.
		 *     logger(payloadType := LogPayloadType.Numeric, numericValue := dev.speedRef, level := LogLevel.DEBUG);
		 *     logger(payloadType := LogPayloadType.Numeric, numericValue := dev.outletColdGlycolTemp, level := LogLevel.DEBUG);
		 *     (* etc. *)
		 *)
	*)
	END_FUNCTION_BLOCK

(* ---- OutputSignalUpdate.pou ---- *)
(*#-#-#-#-#-#-#-#-#-#---Declaration---#-#-#-#-#-#-#-#-#-#-#-#-#*)

{attribute 'no_assign'}
(*
 * Output signals processing (e.g.: debouncing filter) and actuation unit.
 * Map logical output parameters on their physical counterpart, performing processing if necessary.
 *)
FUNCTION_BLOCK OutputSignalUpdate
VAR_EXTERNAL
	dev : DeviceFacade;
	io : IOFacade;
END_VAR
VAR_INPUT
	operationType : OperatingMode;
END_VAR
VAR
	(* Logger facade *)
	logger : LoggerFacade;
END_VAR

(*#-#-#-#-#-#-#-#-#-#---Implementation---#-#-#-#-#-#-#-#-#-#-#-#-#*)

(* Logger facade init *)
logger.enable := TRUE; logger.loggerName := 'OutputSignalUpdate';

logger(message := 'Output signals processing and actuation.', level := LogLevel.DEBUG);

(*
	Logical to physical terminals mapping example:

	IF operationType = OperatingMode.Init THEN
		(* Special processing for the init phase, if needed, such as the restart phase after a blackout. *)
		(* etc. *)
	ELSIF operationType = OperatingMode.Run THEN
		(* For continuous speed values mapping ... *)
		(* Example mapping of a word analog signal *)
		io.speedRefSignal := TO_WORD(dev.speedRef);
		(* Example mapping of a 32-bit analog signal *)
		io.speedRefSignal := realToWordArray(dev.speedRef);
		(* Example mapping of a 64-bit analog signal *)
		io.speedRefSignal := longRealToWordArray(dev.speedRef);
		io.coldGlycolTempSignal := TO_WORD(dev.inletColdGlycolTemp);
		(* Scaling and limiting example *)
		processAnalogOutput(dev.tempSetpoint, 4, 20, dev..tempMin,
			dev.tempMax, 0, 1, 0, wordAnalogOutput => io.tempSetpointSignal);
		(* Drive control word and reference mapping *)
		processDriveCyclicOutData(DriveModel.ABBACH580, dev.compressor.enable, reset := FALSE,
			controlWord => io.compressorControlWord);
		(* Reverse logic *)
		io.condenserFanEnableContactor := NOT condenserFan.enable;
		io.coldGlycolPumpContactor := dev.coldGlycolPump.enable;
		io.coldGlycolPumpContactor := NOT dev.coldGlycolPump.disable;
		io.faultLight := coldGlycolPump.fault;
		...
	END_IF;

	(*
	 * Configure and call the logger facade to log signals where needed.
	 *     logger(payloadType := LogPayloadType.Numeric, numericValue := io.speedRefSignal, level := LogLevel.DEBUG);
	 *     logger(payloadType := LogPayloadType.Numeric, numericValue := io.coldGlycolTempSignal, level := LogLevel.DEBUG);
	 *     logger(payloadType := LogPayloadType.Enum, enumValue := io.controlWord, level := LogLevel.DEBUG);
	 *     (* etc. *)
	 *)
*)

(* ---- OutputSignalUpdate.st ---- *)
(*
 * Output signals processing (e.g.: debouncing filter) and actuation unit.
 * Map logical output parameters on their physical counterpart, performing processing if necessary.
 *)
FUNCTION_BLOCK OutputSignalUpdate
	VAR_EXTERNAL CONSTANT
		applicationDeviceId : STRING;
	END_VAR
	VAR_EXTERNAL
		dev : DeviceFacade;
		io : IOFacade;
	END_VAR
	VAR_INPUT
		operationType : OperatingMode;
	END_VAR
	VAR
		(* Logger facade *)
		logger : LoggerFacade;
	END_VAR

	(* Logger facade init *)
	logger.enable := TRUE; logger.loggerName := applicationDeviceId;

	logger(message := 'Output signals processing and actuation.', level := LogLevel.DEBUG);

	(*
		Logical to physical terminals mapping example:

		IF operationType = OperatingMode.Init THEN
			(* Special processing for the init phase, if needed, such as the restart phase after a blackout. *)
			(* etc. *)
		ELSIF operationType = OperatingMode.Run THEN
			(* For continuous speed values mapping ... *)
			(* Example mapping of a word analog signal *)
			io.speedRefSignal := TO_WORD(dev.speedRef);
			(* Example mapping of a 32-bit analog signal *)
			io.speedRefSignal := realToWordArray(dev.speedRef);
			(* Example mapping of a 64-bit analog signal *)
			io.speedRefSignal := longRealToWordArray(dev.speedRef);
			io.coldGlycolTempSignal := TO_WORD(dev.inletColdGlycolTemp);
			(* Scaling and limiting example *)
			processAnalogOutput(dev.tempSetpoint, 4, 20, dev..tempMin,
				dev.tempMax, 0, 1, 0, wordAnalogOutput => io.tempSetpointSignal);
			(* Drive control word and reference mapping *)
			processDriveCyclicOutData(DriveModel.ABBACH580, dev.compressor.enable, reset := FALSE,
				controlWord => io.compressorControlWord);
			(* Reverse logic *)
			io.condenserFanEnableContactor := NOT condenserFan.enable;
			io.coldGlycolPumpContactor := dev.coldGlycolPump.enable;
			io.coldGlycolPumpContactor := NOT dev.coldGlycolPump.disable;
			io.faultLight := coldGlycolPump.fault;
			...
		END_IF;

		(*
		 * Configure and call the logger facade to log signals where needed.
		 *     logger(payloadType := LogPayloadType.Numeric, numericValue := io.speedRefSignal, level := LogLevel.DEBUG);
		 *     logger(payloadType := LogPayloadType.Numeric, numericValue := io.coldGlycolTempSignal, level := LogLevel.DEBUG);
		 *     logger(payloadType := LogPayloadType.Enum, enumValue := io.controlWord, level := LogLevel.DEBUG);
		 *     (* etc. *)
		 *)
	*)
	END_FUNCTION_BLOCK
